FUNCTION Bind : BoolValue
VAR_INPUT
	boolean : REFERENCE TO BOOL;
END_VAR
VAR
	p : POINTER TO BoolBindingReadOnly;
END_VAR

p := __NEW(BoolBindingReadOnly);

p^.Bind(boolean);

Bind := p^;

END_FUNCTION

(* stored: Version 1.1.0.1
   POU Bind: Id {90e98975-5217-4b6e-97cc-fa4c6cc2a31b}, SpecialFunc None *)
